TYPE SyncUnitsBase_AD6C35CE : STRUCT
END_STRUCT
END_TYPE

(* stored: Version 1.1.0.1, ProductVersion 3.1.4024.11
   DUT SyncUnitsBase_AD6C35CE: Id {4f054d25-c376-026f-2577-d001165e1708} *)
